Universal Robots PolyScope program: lab1_wray_gene.urp

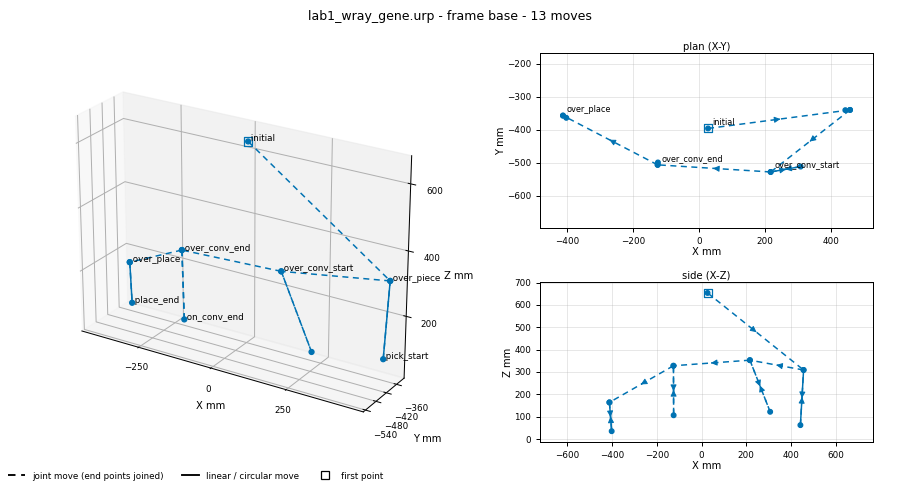
[picture p0: tool path of lab1_wray_gene.urp in frame base, 13 of 13 moves have a stored position in this frame; points joined in program order, loops and branches not executed]
Program lab1_wray_gene (installation=default directory=/programs createdIn=5.14.5 lastSavedIn=5.14.5 robotSerialNumber=20195300809)
Calibrated DH parameters: a=[-0.000085, -0.20076, -0.212369, 0.000121, -0.000118, 0]; d=[0.15185, -26.306375, 24.753047, 1.684739, 0.085386, 0.092088]; alpha=[1.572149, -0.00522, -0.011864, 1.571339, -1.571085, 0]; deltaTheta=[0, 0.599885, -0.513355, -0.086555, 0.000006, 0]
InitVariablesNode
Robot Program (runOnlyOnce=false)
  MoveJ speed 60 deg/s, acceleration 80 deg/s^2 (useActiveTCP=true) feature=Base
    Waypoint initial: TCP in base x=26.788 y=-395.903 z=653.368 mm, rx=0.3299 ry=2.0112 rz=-1.9616 rad; joints [6.184, -70.482, -45.192, -53.231, -3.562, 11.063] deg; TCP offset x=0 y=0 z=174 mm, rx=0 ry=0 rz=0 rad
    URCap Gripper (Robotiq_Grippers, Robotiq Inc.) dataModel(position=0.0, force=0.0, speed=0.0, positionInDouble=0.0, forceInDouble=0.0, speedInDouble=0.0, slaveIds=[9], blocking=true)
    Waypoint over_piece: TCP in base x=456.226 y=-339.878 z=308.82 mm, rx=1.6876 ry=0.0702 rz=0.1151 rad; joints [7.112, -117.978, -66.297, -91.93, 6.01, -81.739] deg; TCP offset x=0 y=0 z=174 mm, rx=0 ry=0 rz=0 rad
    MoveL speed 250 mm/s, acceleration 1200 mm/s^2 (useActiveTCP=true) feature=Base
      Waypoint pick_start: TCP in base x=441.988 y=-340.677 z=62.207 mm, rx=1.6327 ry=0.1187 rz=0.0202 rad; joints [7.401, -144.513, -84.521, -77.422, 3.875, -56.854] deg; TCP offset x=0 y=0 z=174 mm, rx=0 ry=0 rz=0 rad
    URCap Gripper (Robotiq_Grippers, Robotiq Inc.) dataModel(position=100.0, force=0.0, speed=0.0, positionInDouble=100.0, forceInDouble=0.0, speedInDouble=0.0, slaveIds=[9], blocking=true)
    Waypoint over_piece: TCP in base x=456.226 y=-339.878 z=308.82 mm, rx=1.6876 ry=0.0702 rz=0.1151 rad; joints [7.112, -117.978, -66.297, -91.93, 6.01, -81.739] deg; TCP offset x=0 y=0 z=174 mm, rx=0 ry=0 rz=0 rad
    Waypoint over_conv_start: TCP in base x=216.165 y=-527.59 z=352.712 mm, rx=1.4718 ry=-0.3577 rz=-0.2627 rad; joints [-23.858, -116.838, -68.757, -91.239, -4.289, -78.88] deg; TCP offset x=0 y=0 z=174 mm, rx=0 ry=0 rz=0 rad
    Waypoint on_conv_start: TCP in base x=306.751 y=-511.346 z=121.85 mm, rx=1.6208 ry=-0.2137 rz=-0.2893 rad; joints [-17.52, -144.898, -72.497, -68.728, 2.563, -77.128] deg; TCP offset x=0 y=0 z=174 mm, rx=0 ry=0 rz=0 rad
    URCap Gripper (Robotiq_Grippers, Robotiq Inc.) dataModel(position=0.0, force=0.0, speed=0.0, positionInDouble=0.0, forceInDouble=0.0, speedInDouble=0.0, slaveIds=[9], blocking=true)
    MoveJ speed 60 deg/s, acceleration 80 deg/s^2 (useActiveTCP=true) feature=Base
      Waypoint over_conv_start: TCP in base x=216.165 y=-527.59 z=352.712 mm, rx=1.4718 ry=-0.3577 rz=-0.2627 rad; joints [-23.858, -116.838, -68.757, -91.239, -4.289, -78.88] deg; TCP offset x=0 y=0 z=174 mm, rx=0 ry=0 rz=0 rad
    Set DigitalOutput pin=digital_out[0]; digitalValue=1
    Wait DigitalInput pin=digital_in[0]; digitalValue=0
    Set DigitalOutput pin=digital_out[0]; digitalValue=0
    Waypoint over_conv_end: TCP in base x=-125.699 y=-506.046 z=327.792 mm, rx=-0.4485 ry=1.9278 rz=-1.9971 rad; joints [26.325, -77.506, 98.744, -114.248, 1.293, -86.899] deg; TCP offset x=0 y=0 z=174 mm, rx=0 ry=0 rz=0 rad
    MoveJ speed 60 deg/s, acceleration 80 deg/s^2 (useActiveTCP=true) feature=Base
      Waypoint on_conv_end: TCP in base x=-124.883 y=-498.827 z=106.311 mm, rx=-0.4186 ry=1.9878 rz=-1.9648 rad; joints [25.392, -42.418, 116.78, -162.332, -0.795, -91.038] deg
    URCap Gripper (Robotiq_Grippers, Robotiq Inc.) dataModel(position=100.0, force=0.0, speed=0.0, positionInDouble=100.0, forceInDouble=0.0, speedInDouble=0.0, slaveIds=[9], blocking=true)
    Waypoint over_conv_end: TCP in base x=-125.699 y=-506.046 z=327.792 mm, rx=-0.4485 ry=1.9278 rz=-1.9971 rad; joints [26.325, -77.506, 98.744, -114.248, 1.293, -86.899] deg
    Waypoint over_place: TCP in base x=-412.089 y=-357.026 z=163.898 mm, rx=-0.0889 ry=-2.1721 rz=2.1133 rad; joints [-5.811, -46.24, 103.101, -160.652, -2.044, -78.373] deg; TCP offset x=0 y=0 z=174 mm, rx=0 ry=0 rz=0 rad
    Waypoint place_end: TCP in base x=-401.973 y=-363.819 z=35.087 mm, rx=-0.1066 ry=-2.248 rz=2.0569 rad; joints [-4.693, -22.634, 98.44, -178.527, -5.476, -78.449] deg; TCP offset x=0 y=0 z=174 mm, rx=0 ry=0 rz=0 rad
    URCap Gripper (Robotiq_Grippers, Robotiq Inc.) dataModel(position=0.0, force=0.0, speed=0.0, positionInDouble=0.0, forceInDouble=0.0, speedInDouble=0.0, slaveIds=[9], blocking=true)
    MoveL speed 250 mm/s, acceleration 1200 mm/s^2 (useActiveTCP=true) feature=Base
      Waypoint over_place: TCP in base x=-412.089 y=-357.026 z=163.898 mm, rx=-0.0889 ry=-2.1721 rz=2.1133 rad; joints [-5.811, -46.24, 103.101, -160.652, -2.044, -78.373] deg; TCP offset x=0 y=0 z=174 mm, rx=0 ry=0 rz=0 rad
